PROGRAM MAIN
VAR
END_VAR

END_PROGRAM

(* stored: Version 1.1.0.1
   POU MAIN: Id {b245f8ee-2ee0-404f-a6e1-23510d042c82} *)
